FUNCTION_BLOCK TurnOnCommand EXTENDS I_Command
VAR
	_device	:I_Device;
END_VAR

METHOD execute
_device.turnOn();
END_METHOD

METHOD FB_init : BOOL
VAR_INPUT
	bInitRetains : BOOL; // if TRUE, the retain variables are initialized (warm start / cold start)
	bInCopyCode : BOOL;  // if TRUE, the instance afterwards gets moved into the copy code (online change)
	
	device	:I_Device;
END_VAR
This^._device := device;
END_METHOD

END_FUNCTION_BLOCK

(* stored: Version 1.1.0.1, ProductVersion 3.1.4024.12
   POU TurnOnCommand: Id {dc1be576-2ffb-4fa4-af5e-668775f5a935}, SpecialFunc None
   Method execute: Id {be89d116-5d31-405e-a9b4-60cc55fd61f1}
   Method FB_init: Id {6dee32ed-6b33-4bc2-a52e-7d07c51062bd} *)
